FUNCTION_BLOCK FB_UseExtSetpointGen

VAR_INPUT
	Enable :BOOL; // allows motion commands, turn off to disable servo and engage brakes. don't do this while moving unless you don't want to control the decelleration ramp.
	Setpoint_Interface : Setpoint_Interface; // takes values in from the SP gen
END_VAR

VAR
	MC_ExternalSetpointGenEnable :MC_ExtSetPointGenEnable;
	MC_ExternalSetpointGenDisable :MC_ExtSetPointGenDisable;
	ErrorId: UDINT;
END_VAR

VAR_OUTPUT
	Error: BOOL;
	Enabled: BOOL;
	Busy: BOOL;
END_VAR

VAR_IN_OUT
Axis: AXIS_REF; // axis to manipulate	
END_VAR

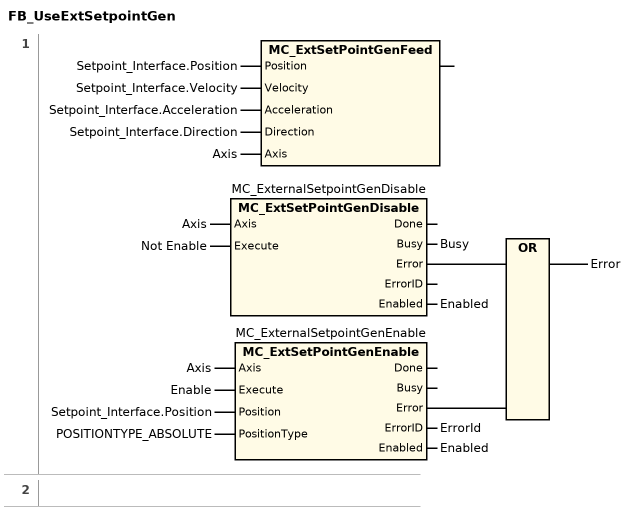
// NETWORK 1
MC_ExtSetPointGenFeed(Position := Setpoint_Interface.Position, Velocity := Setpoint_Interface.Velocity, Acceleration := Setpoint_Interface.Acceleration, Direction := Setpoint_Interface.Direction, Axis := Axis);
MC_ExternalSetpointGenDisable(Axis := Axis, Execute := Not Enable, Busy => Busy, Enabled => Enabled); // MC_ExtSetPointGenDisable
MC_ExternalSetpointGenEnable(
    Axis := Axis,
    Execute := Enable,
    Position := Setpoint_Interface.Position,
    PositionType := POSITIONTYPE_ABSOLUTE,
    ErrorID => ErrorId,
    Enabled => Enabled); // MC_ExtSetPointGenEnable
Error := MC_ExternalSetpointGenDisable.Error OR MC_ExternalSetpointGenEnable.Error;

// NETWORK 2

END_FUNCTION_BLOCK

(* stored: Version 1.1.0.1, ProductVersion 3.1.4024.3
   POU FB_UseExtSetpointGen: Id {2c99fab1-4db1-4e5a-a1fd-36cb2f1d35be}, SpecialFunc None *)
